(* IEC 61131-3 sources: virtual-plc/crates/plc-compiler/fuzz/corpus/fuzz_compile, 4 files *)

(* ---- blink.st ---- *)
(*
 * blink.st - Simple LED blink example
 *
 * This program toggles a digital output at a configurable interval,
 * demonstrating basic timing logic in IEC 61131-3 Structured Text.
 *
 * In a real PLC, this would drive an indicator LED or pilot light.
 * Assuming a 10ms cycle time, this blinks at ~1 Hz (50 cycles on, 50 off).
 *
 * Note: This example uses cycle counting for timing. In production code,
 * you would typically use TON/TOF timer function blocks when available.
 *)

PROGRAM Blink
VAR
    (* Output to LED - would be mapped to hardware via I/O configuration *)
    led_output : BOOL := FALSE;

    (* Cycle counter for timing *)
    counter : INT := 0;

    (* Number of cycles for half-period (50 = 500ms at 10ms cycle) *)
    half_period : INT := 50;
END_VAR

(* Increment counter each scan cycle *)
counter := counter + 1;

(* When counter reaches half_period, toggle LED and reset *)
IF counter >= half_period THEN
    led_output := NOT led_output;
    counter := 0;
END_IF;

END_PROGRAM

(* ---- motor_control.st ---- *)
(*
 * motor_control.st - Motor start/stop with safety interlocks
 *
 * This program demonstrates a typical industrial motor control pattern
 * with start/stop buttons, emergency stop, and safety interlocks.
 *
 * Safety Philosophy:
 *   - Stop button and E-Stop use NC (normally closed) contacts
 *   - Loss of signal = safe state (motor stops)
 *   - Faults are latched until manually reset
 *
 * Variables represent I/O that would be mapped to hardware:
 *   Inputs: start_button, stop_button, e_stop, overload_ok, guard_closed
 *   Outputs: motor_contactor, run_indicator, fault_indicator
 *)

PROGRAM MotorControl
VAR
    (* Inputs - would be mapped to physical I/O *)
    start_button : BOOL := FALSE;   (* Momentary NO - TRUE when pressed *)
    stop_button : BOOL := TRUE;     (* NC - FALSE when pressed (fail-safe) *)
    e_stop : BOOL := TRUE;          (* NC - FALSE when pressed (fail-safe) *)
    overload_ok : BOOL := TRUE;     (* NC - FALSE when tripped *)
    guard_closed : BOOL := TRUE;    (* NO - TRUE when guard is closed *)

    (* Outputs - would be mapped to physical I/O *)
    motor_contactor : BOOL := FALSE;
    run_indicator : BOOL := FALSE;
    fault_indicator : BOOL := FALSE;

    (* Internal state *)
    motor_running : BOOL := FALSE;
    fault_latched : BOOL := FALSE;

    (* Restart delay counter (cycles) - prevents rapid restart *)
    restart_delay_counter : INT := 0;
    restart_delay_target : INT := 200;  (* 2 seconds at 10ms cycle *)
    restart_allowed : BOOL := FALSE;

    (* Composite safety status *)
    safety_ok : BOOL := FALSE;
END_VAR

(* Check all safety interlocks - all must be TRUE for safe operation *)
safety_ok := stop_button AND e_stop AND overload_ok AND guard_closed;

(* Fault detection - latch any fault condition that occurs while running *)
IF NOT safety_ok AND motor_running THEN
    fault_latched := TRUE;
END_IF;

(* Reset fault when conditions are safe and motor is stopped and start not pressed *)
IF NOT motor_running AND safety_ok AND NOT start_button THEN
    fault_latched := FALSE;
END_IF;

(* Restart delay - count up when motor stopped, reset when running *)
IF motor_running THEN
    restart_delay_counter := 0;
    restart_allowed := FALSE;
ELSE
    IF restart_delay_counter < restart_delay_target THEN
        restart_delay_counter := restart_delay_counter + 1;
        restart_allowed := FALSE;
    ELSE
        restart_allowed := TRUE;
    END_IF;
END_IF;

(* Motor start/stop logic - seal-in circuit pattern *)
IF motor_running THEN
    (* Stop conditions: loss of any safety interlock *)
    IF NOT safety_ok THEN
        motor_running := FALSE;
    END_IF;
ELSE
    (* Start conditions: start button + all interlocks + no fault + delay complete *)
    IF start_button AND safety_ok AND NOT fault_latched AND restart_allowed THEN
        motor_running := TRUE;
    END_IF;
END_IF;

(* Update outputs *)
motor_contactor := motor_running;
run_indicator := motor_running;
fault_indicator := fault_latched;

END_PROGRAM

(* ---- pid_control.st ---- *)
(*
 * pid_control.st - PID temperature control example
 *
 * This program demonstrates a basic PID (Proportional-Integral-Derivative)
 * controller for temperature regulation. It includes:
 *
 * - Configurable setpoint and PID gains
 * - Auto/Manual mode switching with bumpless transfer
 * - Output limiting (0-100%)
 * - Anti-windup for integral term (clamping + back-calculation)
 * - Derivative filtering to reduce noise sensitivity
 *
 * Scaling: All values use 0-10000 = 0-100.0 (one decimal place precision)
 * This integer-only implementation avoids floating-point for determinism.
 *)

PROGRAM TemperaturePID
VAR
    (* Inputs - would be mapped to analog I/O *)
    process_value : INT := 5000;      (* Temperature PV, 0-10000 = 0-100.0 C *)
    setpoint_input : INT := 5000;     (* Setpoint, 0-10000 = 0-100.0 C *)
    auto_mode : BOOL := TRUE;         (* TRUE = Auto, FALSE = Manual *)
    manual_output : INT := 0;         (* Manual output 0-10000 = 0-100% *)
    enable : BOOL := TRUE;            (* Controller enable *)

    (* Outputs - would be mapped to analog I/O *)
    control_output : INT := 0;        (* Output to heater, 0-10000 = 0-100% *)
    at_setpoint : BOOL := FALSE;      (* Within deadband of setpoint *)
    high_alarm : BOOL := FALSE;       (* Temperature high alarm *)
    low_alarm : BOOL := FALSE;        (* Temperature low alarm *)

    (* PID Parameters - scaled by 100 for integer math *)
    kp : INT := 200;      (* Proportional gain * 100 (2.0) *)
    ki : INT := 50;       (* Integral gain * 100 (0.5) *)
    kd : INT := 100;      (* Derivative gain * 100 (1.0) *)

    (* Output limits *)
    output_min : INT := 0;
    output_max : INT := 10000;

    (* Integral limits (anti-windup) *)
    integral_min : INT := -5000;
    integral_max : INT := 5000;

    (* Alarm thresholds *)
    high_alarm_sp : INT := 9000;   (* 90.0 C *)
    low_alarm_sp : INT := 1000;    (* 10.0 C *)
    deadband : INT := 50;          (* 0.5 C deadband for "at setpoint" *)

    (* Internal PID state *)
    error : INT := 0;
    error_prev : INT := 0;
    integral : INT := 0;
    derivative : INT := 0;
    derivative_filtered : INT := 0;

    (* Derivative filter coefficient (0-100, higher = more filtering) *)
    derivative_filter : INT := 80;

    (* Working variables *)
    pid_output : INT := 0;
    final_output : INT := 0;
    active_setpoint : INT := 5000;
END_VAR

(* Use external setpoint if valid, otherwise use default *)
IF setpoint_input >= 0 AND setpoint_input <= 10000 THEN
    active_setpoint := setpoint_input;
END_IF;

(* Calculate error: positive = need more heat *)
error := active_setpoint - process_value;

(* Check if controller is enabled *)
IF enable AND auto_mode THEN
    (* === PROPORTIONAL TERM === *)
    (* P = Kp * Error / 100 (done in final calculation) *)

    (* === INTEGRAL TERM with anti-windup === *)
    integral := integral + (ki * error / 1000);

    (* Clamp integral to prevent windup *)
    IF integral > integral_max THEN
        integral := integral_max;
    ELSIF integral < integral_min THEN
        integral := integral_min;
    END_IF;

    (* === DERIVATIVE TERM with filtering === *)
    (* Raw derivative (rate of change of error) *)
    derivative := error - error_prev;

    (* First-order low-pass filter reduces noise sensitivity *)
    (* Filtered = (filter * prev + (100-filter) * raw) / 100 *)
    derivative_filtered := (derivative_filter * derivative_filtered +
                           (100 - derivative_filter) * derivative) / 100;

    (* === CALCULATE PID OUTPUT === *)
    pid_output := (kp * error / 100) + integral + (kd * derivative_filtered / 100);

    (* Bias at 50% - typical for heating-only system *)
    pid_output := pid_output + 5000;

    (* === OUTPUT LIMITING with back-calculation anti-windup === *)
    IF pid_output > output_max THEN
        final_output := output_max;
        (* Back-calculate: undo integral contribution that caused saturation *)
        IF error > 0 THEN
            integral := integral - (ki * error / 1000);
        END_IF;
    ELSIF pid_output < output_min THEN
        final_output := output_min;
        IF error < 0 THEN
            integral := integral - (ki * error / 1000);
        END_IF;
    ELSE
        final_output := pid_output;
    END_IF;

    (* Store previous error for next derivative calculation *)
    error_prev := error;

ELSIF enable AND NOT auto_mode THEN
    (* === MANUAL MODE === *)
    IF manual_output >= output_min AND manual_output <= output_max THEN
        final_output := manual_output;
    END_IF;

    (* Reset integral for bumpless transfer back to auto *)
    integral := 0;
    error_prev := error;

ELSE
    (* === DISABLED - safe state === *)
    final_output := 0;
    integral := 0;
    error_prev := 0;
    derivative_filtered := 0;
END_IF;

(* Update output *)
control_output := final_output;

(* === STATUS OUTPUTS === *)
(* At setpoint if within deadband *)
IF error > -deadband AND error < deadband THEN
    at_setpoint := TRUE;
ELSE
    at_setpoint := FALSE;
END_IF;

(* Alarm outputs *)
high_alarm := process_value > high_alarm_sp;
low_alarm := process_value < low_alarm_sp;

END_PROGRAM

(* ---- state_machine.st ---- *)
(*
 * state_machine.st - Sequential process control (batch mixing example)
 *
 * This program demonstrates a state machine pattern for sequential
 * process control, simulating a simple batch mixing operation:
 *
 * States:
 *   0 = IDLE     - Wait for start command
 *   1 = FILL     - Fill tank to high level
 *   2 = MIX      - Run mixer for specified time
 *   3 = HEAT     - Heat to target temperature
 *   4 = DRAIN    - Drain tank to low level
 *   5 = COMPLETE - Signal done, return to IDLE
 *
 * This pattern is common in batch processing, packaging, and assembly operations.
 *)

PROGRAM BatchMixer
VAR
    (* State constants *)
    STATE_IDLE : INT := 0;
    STATE_FILL : INT := 1;
    STATE_MIX : INT := 2;
    STATE_HEAT : INT := 3;
    STATE_DRAIN : INT := 4;
    STATE_COMPLETE : INT := 5;

    (* Current state *)
    current_state : INT := 0;

    (* Inputs - would be mapped to physical I/O *)
    start_batch : BOOL := FALSE;      (* Start command from HMI/button *)
    tank_low : BOOL := TRUE;          (* Low level sensor - TRUE when below low *)
    tank_high : BOOL := FALSE;        (* High level sensor - TRUE when above high *)
    temperature : INT := 200;         (* Temperature sensor 0-1000 = 0-100.0 C *)
    e_stop : BOOL := TRUE;            (* Emergency stop NC - FALSE when pressed *)

    (* Outputs - would be mapped to physical I/O *)
    fill_valve : BOOL := FALSE;
    drain_valve : BOOL := FALSE;
    mixer_motor : BOOL := FALSE;
    heater : BOOL := FALSE;
    batch_complete : BOOL := FALSE;
    state_output : INT := 0;          (* Current state for HMI display *)

    (* Process parameters *)
    mix_time_cycles : INT := 3000;    (* 30 seconds at 10ms cycle *)
    target_temp : INT := 750;         (* 75.0 C in scaled units *)
    temp_hysteresis : INT := 20;      (* 2.0 C hysteresis *)
    complete_delay : INT := 500;      (* 5 seconds at 10ms cycle *)

    (* Timer counters *)
    mix_counter : INT := 0;
    complete_counter : INT := 0;
END_VAR

(* Emergency stop handling - immediate safe shutdown *)
IF NOT e_stop THEN
    current_state := STATE_IDLE;
    fill_valve := FALSE;
    drain_valve := FALSE;
    mixer_motor := FALSE;
    heater := FALSE;
    batch_complete := FALSE;
    mix_counter := 0;
    complete_counter := 0;
END_IF;

(* State machine - CASE statement is ideal for sequential control *)
CASE current_state OF
    0: (* IDLE - Safe state, all outputs off *)
        fill_valve := FALSE;
        drain_valve := FALSE;
        mixer_motor := FALSE;
        heater := FALSE;
        batch_complete := FALSE;
        mix_counter := 0;
        complete_counter := 0;

        (* Start only if e-stop OK and tank is empty *)
        IF start_batch AND e_stop AND tank_low THEN
            current_state := STATE_FILL;
        END_IF;

    1: (* FILL - Open fill valve until high level *)
        fill_valve := TRUE;
        drain_valve := FALSE;

        IF tank_high THEN
            fill_valve := FALSE;
            current_state := STATE_MIX;
        END_IF;

    2: (* MIX - Run mixer for specified time *)
        mixer_motor := TRUE;
        mix_counter := mix_counter + 1;

        IF mix_counter >= mix_time_cycles THEN
            mix_counter := 0;
            current_state := STATE_HEAT;
        END_IF;

    3: (* HEAT - Heat with temperature control *)
        mixer_motor := TRUE;  (* Keep mixing while heating *)

        (* Bang-bang control with hysteresis *)
        IF temperature < target_temp - temp_hysteresis THEN
            heater := TRUE;
        ELSIF temperature >= target_temp THEN
            heater := FALSE;
            current_state := STATE_DRAIN;
        END_IF;

    4: (* DRAIN - Open drain valve until empty *)
        mixer_motor := FALSE;
        heater := FALSE;
        drain_valve := TRUE;

        IF tank_low THEN
            drain_valve := FALSE;
            current_state := STATE_COMPLETE;
        END_IF;

    5: (* COMPLETE - Signal done, delay, return to IDLE *)
        batch_complete := TRUE;
        complete_counter := complete_counter + 1;

        IF complete_counter >= complete_delay THEN
            complete_counter := 0;
            batch_complete := FALSE;
            current_state := STATE_IDLE;
        END_IF;
END_CASE;

(* Output current state for HMI display *)
state_output := current_state;

END_PROGRAM
